ADAPTER IFlushReady (* Adapter Interface *)
  (* Standard: 61499-1 *)
  (* Version 0.0, 7/21/2026, Schneider Electric *)
  PACKAGE SE.Nereda;
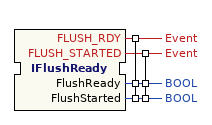
  EVENT_OUTPUT
    FLUSH_RDY WITH FlushReady, FlushStarted; (* Confirmation from Plug *)
    FLUSH_STARTED WITH FlushStarted, FlushReady;
  END_EVENT
  VAR_OUTPUT
    FlushReady : BOOL; (* Confirmation Data from Plug *)
    FlushStarted : BOOL;
  END_VAR
  SERVICE SOCKET/PLUG
    SEQUENCE request_confirm
      SOCKET.REQ(REQD) -> PLUG.REQ(REQD);
      PLUG.FLUSH_RDY(FlushReady) -> SOCKET.FLUSH_RDY(FlushReady);
    END_SEQUENCE
    SEQUENCE indication_response
      PLUG.IND(INDD) -> SOCKET.IND(INDD);
      SOCKET.RSP(RSPD) -> PLUG.RSP(RSPD);
    END_SEQUENCE
  END_SERVICE
END_ADAPTER
